PROGRAM main
VAR
	//sensori
	SensoreStart : BOOL := FALSE;
	SensoreReset : BOOL := FALSE;
	SensoreFCBottom : BOOL := FALSE;
	SensoreFCTop : BOOL := FALSE;
	SensoreFCS : BOOL := FALSE;
	SensoreFCD : BOOL := FALSE;
	SensoreFCP : BOOL := FALSE;
	SensoreGrasp : BOOL := FALSE;
	SensoreRelease : BOOL := FALSE;
	SensoreRulloOccupato : BOOL := FALSE;
	SensoreVascaVuota : BOOL := FALSE;
	{attribute 'OPC.UA.DA' := '1'}
	SensoreIsGiorno : BOOL := FALSE;
	SensoreSerbatoioOn : BOOL := FALSE;
	SensoreSerbatoioFull : BOOL := TRUE;
	SensoreSerbatoioEmpty : BOOL := FALSE;
	SensoreCondizionatore : BOOL := FALSE;
	SensoreApriFinestra : BOOL := FALSE;
	SensoreTempCalda : BOOL := FALSE;
	SensoreTempFredda : BOOL := FALSE;
	SensoreO2Low : BOOL := FALSE;
	SensorePianta1Pronta : BOOL := FALSE;
	SensorePianta2Pronta : BOOL := FALSE;
	//attuatori
	AttuatBraccioGiu : BOOL := FALSE;
	AttuatBraccioSu : BOOL := FALSE;
	AttuatBraccioSx : BOOL := FALSE;
	AttuatBraccioDx : BOOL := FALSE;
	AttuatBraccioPresa : BOOL := FALSE;
	AttuatBraccioRilascio : BOOL := FALSE;
	AttuatRiempiSerbatoio : BOOL := FALSE;
	AttuatSvuotaSerbatoio : BOOL := FALSE;
	AttuatFinestra : BOOL := FALSE;
	AttuatCondizionatore : BOOL := FALSE;
	AttuatRullo : BOOL := FALSE;
	AttuatLampada : BOOL := FALSE;
	
	//WatchDog e Allarme
	WatchDog : TON;
	TimerWatchDog : TIME := TIME#10S;
	{attribute 'OPC.UA.DA' := '1'}
	Allarme1 : BOOL := FALSE;
	{attribute 'OPC.UA.DA' := '1'}
	ContatorePiante : INT := 0;
	
	//Variabili RunTime per SCADA
	{attribute 'OPC.UA.DA' := '1'}
	Temperatura : LREAL;
	{attribute 'OPC.UA.DA' := '1'}
	Ossigeno: LREAL;
	
	AggiuntoPianta : BOOL := FALSE;
END_VAR

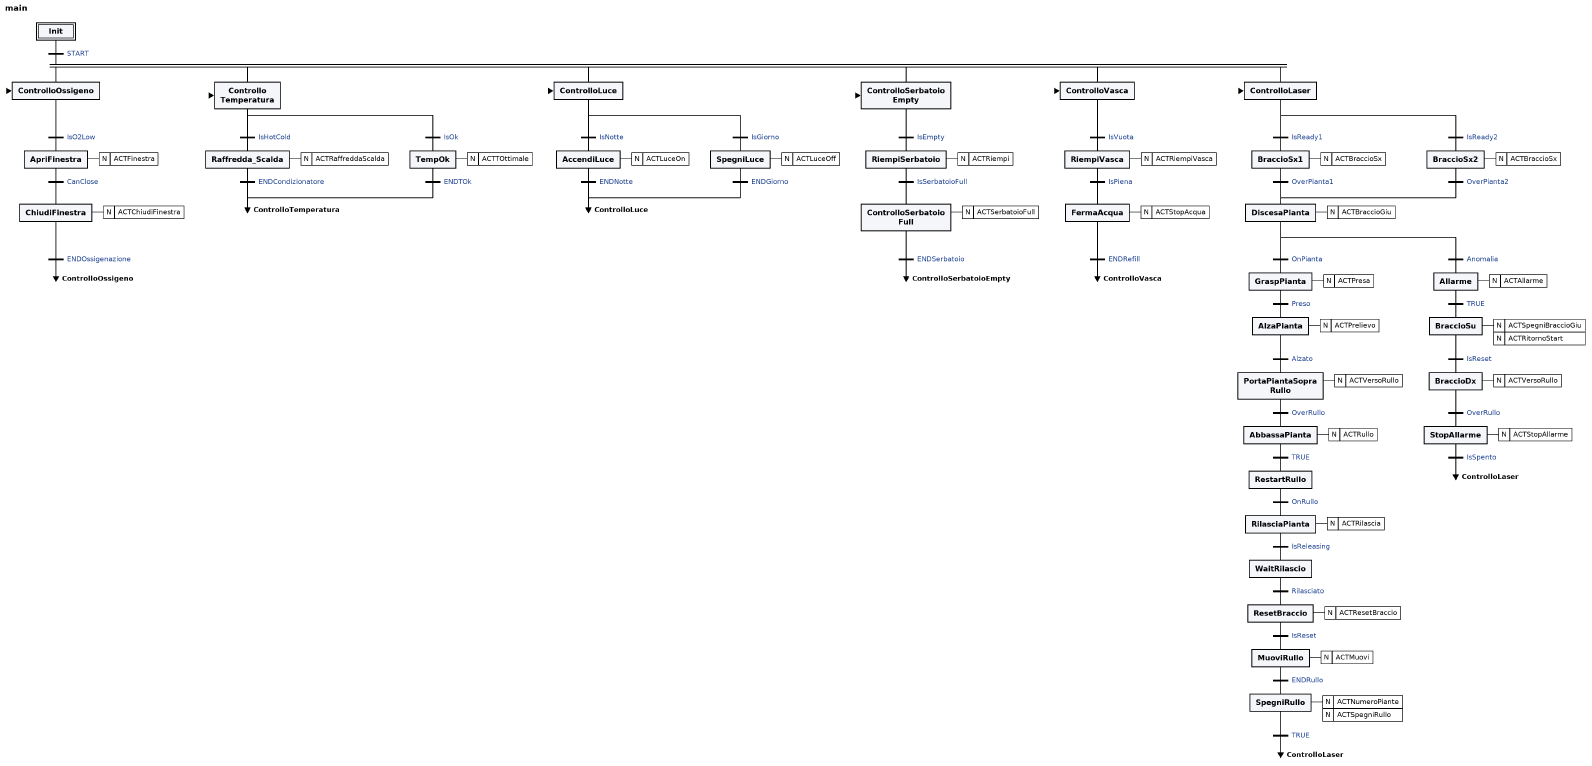
INITIAL_STEP Init:
END_STEP
TRANSITION FROM Init TO (ControlloOssigeno, ControlloTemperatura, ControlloLuce, ControlloSerbatoioEmpty, ControlloVasca, ControlloLaser)
    := START;
END_TRANSITION
STEP ControlloOssigeno:
END_STEP
TRANSITION FROM ControlloOssigeno TO ApriFinestra
    := IsO2Low;
END_TRANSITION
STEP ApriFinestra:
    ACTFinestra(N);
END_STEP
TRANSITION FROM ApriFinestra TO ChiudiFinestra
    := CanClose;
END_TRANSITION
STEP ChiudiFinestra:
    ACTChiudiFinestra(N);
END_STEP
TRANSITION FROM ChiudiFinestra TO ControlloOssigeno
    := ENDOssigenazione;
END_TRANSITION
STEP ControlloTemperatura:
END_STEP
TRANSITION FROM ControlloTemperatura TO Raffredda_Scalda
    := IsHotCold;
END_TRANSITION
STEP Raffredda_Scalda:
    ACTRaffreddaScalda(N);
END_STEP
TRANSITION FROM Raffredda_Scalda TO ControlloTemperatura
    := ENDCondizionatore;
END_TRANSITION
TRANSITION FROM ControlloTemperatura TO TempOk
    := IsOk;
END_TRANSITION
STEP TempOk:
    ACTTOttimale(N);
END_STEP
TRANSITION FROM TempOk TO ControlloTemperatura
    := ENDTOk;
END_TRANSITION
STEP ControlloLuce:
END_STEP
TRANSITION FROM ControlloLuce TO AccendiLuce
    := IsNotte;
END_TRANSITION
STEP AccendiLuce:
    ACTLuceOn(N);
END_STEP
TRANSITION FROM AccendiLuce TO ControlloLuce
    := ENDNotte;
END_TRANSITION
TRANSITION FROM ControlloLuce TO SpegniLuce
    := IsGiorno;
END_TRANSITION
STEP SpegniLuce:
    ACTLuceOff(N);
END_STEP
TRANSITION FROM SpegniLuce TO ControlloLuce
    := ENDGiorno;
END_TRANSITION
STEP ControlloSerbatoioEmpty:
END_STEP
TRANSITION FROM ControlloSerbatoioEmpty TO RiempiSerbatoio
    := IsEmpty;
END_TRANSITION
STEP RiempiSerbatoio:
    ACTRiempi(N);
END_STEP
TRANSITION FROM RiempiSerbatoio TO ControlloSerbatoioFull
    := IsSerbatoioFull;
END_TRANSITION
STEP ControlloSerbatoioFull:
    ACTSerbatoioFull(N);
END_STEP
TRANSITION FROM ControlloSerbatoioFull TO ControlloSerbatoioEmpty
    := ENDSerbatoio;
END_TRANSITION
STEP ControlloVasca:
END_STEP
TRANSITION FROM ControlloVasca TO RiempiVasca
    := IsVuota;
END_TRANSITION
STEP RiempiVasca:
    ACTRiempiVasca(N);
END_STEP
TRANSITION FROM RiempiVasca TO FermaAcqua
    := IsPiena;
END_TRANSITION
STEP FermaAcqua:
    ACTStopAcqua(N);
END_STEP
TRANSITION FROM FermaAcqua TO ControlloVasca
    := ENDRefill;
END_TRANSITION
STEP ControlloLaser:
END_STEP
TRANSITION FROM ControlloLaser TO BraccioSx1
    := IsReady1;
END_TRANSITION
STEP BraccioSx1:
    ACTBraccioSx(N);
END_STEP
TRANSITION FROM BraccioSx1 TO DiscesaPianta
    := OverPianta1;
END_TRANSITION
TRANSITION FROM ControlloLaser TO BraccioSx2
    := IsReady2;
END_TRANSITION
STEP BraccioSx2:
    ACTBraccioSx(N);
END_STEP
TRANSITION FROM BraccioSx2 TO DiscesaPianta
    := OverPianta2;
END_TRANSITION
STEP DiscesaPianta:
    ACTBraccioGiu(N);
END_STEP
TRANSITION FROM DiscesaPianta TO GraspPianta
    := OnPianta;
END_TRANSITION
STEP GraspPianta:
    ACTPresa(N);
END_STEP
TRANSITION FROM GraspPianta TO AlzaPianta
    := Preso;
END_TRANSITION
TRANSITION FROM DiscesaPianta TO Allarme
    := Anomalia;
END_TRANSITION
STEP Allarme:
    ACTAllarme(N);
END_STEP
TRANSITION FROM Allarme TO BraccioSu
    := TRUE;
END_TRANSITION
STEP BraccioSu:
    ACTSpegniBraccioGiu(N);
    ACTRitornoStart(N);
END_STEP
TRANSITION FROM BraccioSu TO BraccioDx
    := IsReset;
END_TRANSITION
STEP BraccioDx:
    ACTVersoRullo(N);
END_STEP
TRANSITION FROM BraccioDx TO StopAllarme
    := OverRullo;
END_TRANSITION
STEP StopAllarme:
    ACTStopAllarme(N);
END_STEP
TRANSITION FROM StopAllarme TO ControlloLaser
    := IsSpento;
END_TRANSITION
STEP AlzaPianta:
    ACTPrelievo(N);
END_STEP
TRANSITION FROM AlzaPianta TO PortaPiantaSopraRullo
    := Alzato;
END_TRANSITION
STEP PortaPiantaSopraRullo:
    ACTVersoRullo(N);
END_STEP
TRANSITION FROM PortaPiantaSopraRullo TO AbbassaPianta
    := OverRullo;
END_TRANSITION
STEP AbbassaPianta:
    ACTRullo(N);
END_STEP
TRANSITION FROM AbbassaPianta TO RestartRullo
    := TRUE;
END_TRANSITION
STEP RestartRullo:
END_STEP
TRANSITION FROM RestartRullo TO RilasciaPianta
    := OnRullo;
END_TRANSITION
STEP RilasciaPianta:
    ACTRilascia(N);
END_STEP
TRANSITION FROM RilasciaPianta TO WaitRilascio
    := IsReleasing;
END_TRANSITION
STEP WaitRilascio:
END_STEP
TRANSITION FROM WaitRilascio TO ResetBraccio
    := Rilasciato;
END_TRANSITION
STEP ResetBraccio:
    ACTResetBraccio(N);
END_STEP
TRANSITION FROM ResetBraccio TO MuoviRullo
    := IsReset;
END_TRANSITION
STEP MuoviRullo:
    ACTMuovi(N);
END_STEP
TRANSITION FROM MuoviRullo TO SpegniRullo
    := ENDRullo;
END_TRANSITION
STEP SpegniRullo:
    ACTNumeroPiante(N);
    ACTSpegniRullo(N);
END_STEP
TRANSITION FROM SpegniRullo TO ControlloLaser
    := TRUE;
END_TRANSITION

ACTION ACTAllarme:
Allarme1 := TRUE;
END_ACTION

ACTION ACTBraccioGiu:
AttuatBraccioSx := FALSE;
AttuatBraccioGiu := TRUE;
WatchDog(IN := TRUE, PT := TimerWatchDog);
END_ACTION

ACTION ACTBraccioSx:
AttuatBraccioSx := TRUE;
END_ACTION

ACTION ACTChiudiFinestra:
AttuatFinestra := FALSE;
END_ACTION

ACTION ACTFinestra:
AttuatFinestra := TRUE;
END_ACTION

ACTION ACTLuceOff:
AttuatLampada := FALSE;
END_ACTION

ACTION ACTLuceOn:
AttuatLampada := TRUE;
END_ACTION

ACTION ACTMuovi:
AttuatBraccioSu := FALSE;
AttuatRullo := TRUE;
END_ACTION

ACTION ACTNumeroPiante:
IF AggiuntoPianta = FALSE THEN
	ContatorePiante := ContatorePiante+1;
	AggiuntoPianta := TRUE;
END_IF
END_ACTION

ACTION ACTPrelievo:
AttuatBraccioPresa := FALSE;
AttuatBraccioSu := TRUE;
END_ACTION

ACTION ACTPresa:
AttuatBraccioGiu := FALSE;
AttuatBraccioPresa := TRUE;
WatchDog(IN := FALSE, PT := TimerWatchDog);
AggiuntoPianta := FALSE;
END_ACTION

ACTION ACTRaffreddaScalda:
//Dovrebbe azionare il condizionare freddo
AttuatCondizionatore := TRUE;
END_ACTION

ACTION ACTResetBraccio:
AttuatBraccioRilascio := FALSE;
AttuatBraccioSu := TRUE;
END_ACTION

ACTION ACTRiempi:
AttuatRiempiSerbatoio := TRUE;
END_ACTION

ACTION ACTRiempiVasca:
AttuatSvuotaSerbatoio := TRUE;
END_ACTION

ACTION ACTRilascia:
AttuatBraccioGiu := FALSE;
AttuatBraccioRilascio := TRUE;
END_ACTION

ACTION ACTRitornoStart:
AttuatBraccioSu := TRUE;
END_ACTION

ACTION ACTRullo:
AttuatBraccioDx := FALSE;
AttuatBracciogiu := TRUE;
END_ACTION

ACTION ACTSerbatoioFull:
AttuatRiempiSerbatoio := FALSE;
END_ACTION

ACTION ACTSpegniBraccioGiu:
AttuatBraccioGiu := FALSE;
END_ACTION

ACTION ACTSpegniRullo:
AttuatRullo := FALSE;
END_ACTION

ACTION ACTStopAcqua:
AttuatSvuotaSerbatoio := FALSE;
END_ACTION

ACTION ACTStopAllarme:
AttuatBraccioDx := FALSE;
Allarme1 := FALSE;
WatchDog(IN := FALSE, PT := TimerWatchDog);
END_ACTION

ACTION ACTTOttimale:
AttuatCondizionatore := FALSE;
END_ACTION

ACTION ACTVersoRullo:
//QUI PUOI MERGIARE
AttuatBraccioSu := FALSE;
AttuatBraccioDx := TRUE;
END_ACTION

TRANSITION Alzato:
SensoreFCTop = TRUE
END_TRANSITION

TRANSITION Anomalia:
WatchDog.Q = TRUE
END_TRANSITION

TRANSITION CanClose:
SensoreApriFinestra = FALSE AND SensoreO2Low = FALSE
END_TRANSITION

TRANSITION ENDCondizionatore:
AttuatCondizionatore = TRUE AND SensoreCondizionatore = TRUE
END_TRANSITION

TRANSITION ENDGiorno:
AttuatLampada = FALSE
END_TRANSITION

TRANSITION ENDNotte:
AttuatLampada = TRUE
END_TRANSITION

TRANSITION ENDOssigenazione:
AttuatFinestra = FALSE
END_TRANSITION

TRANSITION ENDRefill:
AttuatSvuotaSerbatoio = FALSE
END_TRANSITION

TRANSITION ENDRullo:
SensoreRulloOccupato = FALSE
END_TRANSITION

TRANSITION ENDSerbatoio:
AttuatRiempiSerbatoio = FALSE
END_TRANSITION

TRANSITION ENDTOk:
AttuatCondizionatore = FALSE AND SensoreCondizionatore = FALSE
END_TRANSITION

TRANSITION IsEmpty:
SensoreSerbatoioEmpty = TRUE
END_TRANSITION

TRANSITION IsGiorno:
SensoreIsGiorno = TRUE
END_TRANSITION

TRANSITION IsHotCold:
SensoreTempCalda = TRUE OR SensoreTempFredda = TRUE
END_TRANSITION

TRANSITION IsNotte:
SensoreIsGiorno = FALSE
END_TRANSITION

TRANSITION IsO2Low:
SensoreO2Low = TRUE AND SensoreApriFinestra = TRUE
END_TRANSITION

TRANSITION IsOk:
SensoreTempFredda = FALSE AND SensoreTempCalda = FALSE
END_TRANSITION

TRANSITION IsPiena:
SensoreSerbatoioOn = FALSE AND SensoreVascaVuota = FALSE
END_TRANSITION

TRANSITION IsReady1:
SensorePianta1Pronta = TRUE
END_TRANSITION

TRANSITION IsReady2:
SensorePianta2Pronta = TRUE
END_TRANSITION

TRANSITION IsReleasing:
SensoreRelease = TRUE
END_TRANSITION

TRANSITION IsReset:
SensoreFCTop = TRUE
END_TRANSITION

TRANSITION IsSerbatoioFull:
SensoreSerbatoioFull = TRUE
END_TRANSITION

TRANSITION IsSpento:
Allarme1 = FALSE
END_TRANSITION

TRANSITION IsVuota:
 //AND SensoreSerbatoioOn = TRUE
SensoreVascaVuota = TRUE AND SensoreSerbatoioEmpty = FALSE
END_TRANSITION

TRANSITION OnPianta:
SensoreFCBottom = TRUE AND WatchDog.Q = FALSE
END_TRANSITION

TRANSITION OnRullo:
SensoreFCBottom = TRUE AND SensoreRulloOccupato = TRUE
END_TRANSITION

TRANSITION OverPianta1:
SensoreFCS = TRUE
END_TRANSITION

TRANSITION OverPianta2:
SensoreFCP = TRUE
END_TRANSITION

TRANSITION OverRullo:
SensoreFCD = TRUE
END_TRANSITION

TRANSITION Preso:
SensoreGrasp = TRUE
END_TRANSITION

TRANSITION RESTART:
SensoreReset = TRUE
END_TRANSITION

TRANSITION Rilasciato:
SensoreRelease = FALSE
END_TRANSITION

TRANSITION START:
SensoreStart = TRUE AND SensoreFCTop= TRUE AND SensoreFCD = TRUE AND SensoreRulloOccupato = FALSE
END_TRANSITION

END_PROGRAM

(* stored: Version 1.1.0.1, ProductVersion 3.1.4024.15
   POU main: Id {b7796c3c-63d4-40cc-8177-a4d52dd478d6}, SpecialFunc None
   Action ACTAllarme: Id {66457109-4593-4465-96f4-8672b8754f04}
   Action ACTBraccioGiu: Id {76a52fda-215b-4da5-b5b4-ab3a76f4f0e7}
   Action ACTBraccioSx: Id {6e12c1b2-772c-4d81-aebc-3e4ef6fcb0a3}
   Action ACTChiudiFinestra: Id {120c9703-b01e-402e-b11d-49dfce91f14e}
   Action ACTFinestra: Id {a5bb2cba-42b2-4dd7-b48c-a76f9b7f28ed}
   Action ACTLuceOff: Id {b7c0274c-d122-4f95-bb16-53e5dea9700b}
   Action ACTLuceOn: Id {d65456a8-c548-4245-bec8-6f1aa287b576}
   Action ACTMuovi: Id {800b6f22-bd1a-4088-91a2-f9671143c9ea}
   Action ACTNumeroPiante: Id {f2880276-3cc8-44f8-89bd-f88c0e4bed82}
   Action ACTPrelievo: Id {f35df336-bc57-415e-98f9-5457ec708268}
   Action ACTPresa: Id {dab20041-4f8d-4bea-b8e8-6097aeb4d7b9}
   Action ACTRaffreddaScalda: Id {3a65b2f5-722a-4fb2-b207-a127cab396a2}
   Action ACTResetBraccio: Id {5edf422e-664b-400b-adab-4de0d28232f5}
   Action ACTRiempi: Id {51e4f0e2-d1bb-4832-8ee4-332df75dfe34}
   Action ACTRiempiVasca: Id {df8a8a99-0711-4147-b60d-0cbe698a8995}
   Action ACTRilascia: Id {0a01667d-4ddd-4b99-b779-cb2163d5f399}
   Action ACTRitornoStart: Id {4bf86ce4-a296-4532-be64-c67f108d5634}
   Action ACTRullo: Id {6c011d45-bca6-445b-a197-11a81c287d73}
   Action ACTSerbatoioFull: Id {1edc2337-f824-4a82-a983-7ea9b4cf36f8}
   Action ACTSpegniBraccioGiu: Id {8600bdfd-5ff1-49fc-b610-ce8d61973c97}
   Action ACTSpegniRullo: Id {191ae01f-ae4e-4ab3-907b-310d8aaa0c99}
   Action ACTStopAcqua: Id {1ccf8d5e-a673-4819-b8d0-3337833f328d}
   Action ACTStopAllarme: Id {e0a4da6d-8262-49d3-9f1b-751e74b1ebc8}
   Action ACTTOttimale: Id {519471eb-ffb2-4ed3-b156-5af6a0715aca}
   Action ACTVersoRullo: Id {4351d1dc-63a2-4d9e-a1f6-cae15d60eb02}
   Transition Alzato: Id {fd682374-57a2-4f73-90a7-8661417fd125}
   Transition Anomalia: Id {8851ed4f-73c6-4a6c-96d2-3019f4cced69}
   Transition CanClose: Id {c9faa1a5-4a3f-488f-99d5-6d9c289dc914}
   Transition ENDCondizionatore: Id {6fa824dd-dbe2-4fbe-abec-72ac4d906280}
   Transition ENDGiorno: Id {d3b8d1d2-6c66-4298-9cc7-06e1f3cb89ea}
   Transition ENDNotte: Id {51370939-99bc-4964-85d6-01549719c4d7}
   Transition ENDOssigenazione: Id {a5efe17c-fcdd-45b4-8c4a-5d7443d056cf}
   Transition ENDRefill: Id {f0c64860-280c-4649-aff2-d517a07b26aa}
   Transition ENDRullo: Id {431f1e4b-6835-4c70-bac9-98c2446fb5fa}
   Transition ENDSerbatoio: Id {8e039238-1019-4833-85cf-f7294c62ef24}
   Transition ENDTOk: Id {42b27609-606c-4132-ac1e-cafbdddbe866}
   Transition IsEmpty: Id {2a65a6b1-03b3-4cd7-a61b-e398bb4c56ec}
   Transition IsGiorno: Id {e410fac9-7132-45dd-ba4a-2c6cc9549a26}
   Transition IsHotCold: Id {fa3cf8e0-8591-4adf-b11d-d748c3d06fc1}
   Transition IsNotte: Id {5f662753-e781-4753-bc51-0a6da238e930}
   Transition IsO2Low: Id {73fb107d-85bb-4d69-a677-79ec4f3cd344}
   Transition IsOk: Id {94dadf6a-ce5d-498f-980d-b2643ed6d930}
   Transition IsPiena: Id {63e11183-3cf8-47bb-82d5-d9d53dcdc247}
   Transition IsReady1: Id {9e132d8b-2a78-47ee-b282-a7deb61649ab}
   Transition IsReady2: Id {495a7330-993b-43ce-a691-d3eac9d7d9e9}
   Transition IsReleasing: Id {06e84cc4-a324-4061-a4a6-e89336e351a8}
   Transition IsReset: Id {edc9d848-7513-4e8d-b918-294792924c66}
   Transition IsSerbatoioFull: Id {62c3f99a-fb09-407c-a091-4f8ccff5bd38}
   Transition IsSpento: Id {c686a197-5af4-424c-b14f-f4833ca78b8d}
   Transition IsVuota: Id {4b8a749a-f6bf-41b8-a28c-bad04e7416cc}
   Transition OnPianta: Id {9c1dbab7-9789-41cb-ac9e-c6e376fa63e8}
   Transition OnRullo: Id {4cbd4b41-7880-4c10-b48d-e7459f1587c7}
   Transition OverPianta1: Id {a1467582-4930-4043-9a4b-405ad4a4c197}
   Transition OverPianta2: Id {80fbacc1-ba08-4786-8ab3-7172e3cb465c}
   Transition OverRullo: Id {462df9c8-eba7-4dc0-9395-0fac21534f6d}
   Transition Preso: Id {13f12b77-d421-43ca-a67f-0764d3c8f6c2}
   Transition RESTART: Id {05697ece-15c4-43a1-b7af-f483519e869e}
   Transition Rilasciato: Id {2735dd17-faa8-469a-aefe-f797c8c6d803}
   Transition START: Id {58dfda41-c2f0-40b5-97e0-a48c1eae994f} *)
